Staubli VAL3: onStart.pgx

program onStart()
  local num i
  local num l_nIndex
  local bool l_bOk
begin
  // INIT
  sTrajName=sItems
  nView=0
  nIndex=0
  bExit=false
  link(fFather,world)
  call trajType:getFrame(fFather,false)
  // set the index
  l_bOk=true
  if size(sItems)>1 and sItems[1]!=""
    toNum(sItems[1],nIndexItem,l_bOk)
  else
    nIndexItem=0
  endIf
  // empty the userMenu
  for i=0 to size(sMenuUser)-1
    sMenuUser[i]=""
  endFor
  // load the traj type
  call loadEditTraj(sItems)
  //endIf
  //
  // logMsg
  logMsg("[KERNEL] INTERFACE:PAGE Edit TRAJ")
  // reset the Key pressure
  call use:nullKey(nKey)
  // define the list
  call buildList()
  //
end
